// TIA Portal project "Yıldız-Üçgen Uygulaması" (V18)

(* hardware
DEVICE "S7-1200 station_1"  S7-1200 Station
   slot 0: "Rack_0"  S7-1200 Rack  Rack  V1.0
   slot 1: "PLC_1"  CPU 1214C AC/DC/Rly  6ES7 214-1BG40-0XB0  V4.6
*)

// ===== PLC "PLC_1"  CPU 1214C AC/DC/Rly =====

VAR_GLOBAL   // PLC tag table "Default tag table"
   "Stop" AT %I0.0 : Bool;
   "Start" AT %I0.1 : Bool;
   "Yıldız" AT %Q0.0 : Bool;
   "Üçgen" AT %Q0.1 : Bool;
END_VAR

// folder: System blocks/Program resources

DATA_BLOCK "IEC_Timer_0_DB_3"   // DB4
{ S7_Optimized_Access := 'TRUE' }
AUTHOR : Simatic
FAMILY : IEC
NAME : IEC_TMR
VERSION : 1.0
// stored: InstanceOfName IEC_TIMER
"IEC_TIMER"
BEGIN
END_DATA_BLOCK

// folder: (top level)

ORGANIZATION_BLOCK "Main"   // OB1, LAD, ProgramCycle
TITLE = "Main Program Sweep (Cycle)"
{ S7_Optimized_Access := 'TRUE' }
VERSION : 0.1
// Yıldız Üçgen Yol Verme İşlemi
   VAR_INPUT
      Initial_Call : Bool;   // Initial call of this OB
      Remanence : Bool;   // =True, if remanent data are available
   END_VAR
BEGIN

REGION Network 1
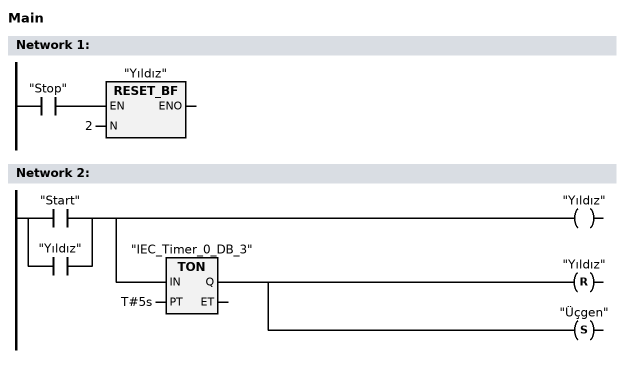
   // no SCL statement known for RBitfield: written as a call
   IF "Stop" THEN RESET_BF(operand := "Yıldız", n := 2); END_IF;
END_REGION

REGION Network 2
   "Yıldız" := "Start" OR "Yıldız";
   "IEC_Timer_0_DB_3".TON(IN := "Yıldız", PT := T#5s);
   IF "IEC_Timer_0_DB_3".Q THEN
       "Yıldız" := FALSE;
       "Üçgen" := TRUE;
   END_IF;
END_REGION
END_ORGANIZATION_BLOCK